PROGRAM Call_Std_Func
VAR
	Start: BOOL;
	Stop: BOOL;
	Motor1: BOOL;
	Motor2: BOOL;
	Timer1: TON;
	Done: BOOL;
	ElapsedTime: TIME;
	Timer2: TON;
END_VAR

IF Start THEN
	Motor1 := TRUE;
END_IF

IF Motor1 THEN
	Timer1(IN:=TRUE , PT:= T#5S, Q=>Done , ET=> ElapsedTime);
END_IF

IF TIMER1.Q THEN
	Timer1(IN := FALSE);
	Motor2 := TRUE;
END_IF

IF Stop THEN
	Motor1 := FALSE;
	Motor2 := FALSE;
END_IF

END_PROGRAM

(* stored: Version 1.1.0.1, ProductVersion 3.1.4024.9
   POU Call_Std_Func: Id {3b1f9f87-2fee-4ed5-8e90-d111f115cc2e}, SpecialFunc None *)
